Staubli VAL3: onF3Event.pgx

program onF3Event()
  local string l_sMessage
begin
  // look if the bButton is enable
  if bButton[2]
    //
  endIf
end
